// SIMATIC STEP 7 (V5.x) project ZEn01_01_STEP7__STL_1-9
// CPU: CPU314(1)
// station: _S7H_BUSSYSTEM_CT
// station: Hardware
// station: SIMATIC 300(1)
// program: S7-Program(1)

SYMBOL_TABLE
"Petrol"	DB 1	FB 1	// Data for petrol engine
"Diesel"	DB 2	FB 1	// Data for diesel engine
"S_Data"	DB 3	DB 3	// Shared data block
"Engine"	FB 1	FB 1	// Engine control
"Fan"	FC 1	FC 1	// Fan control
"Key_1"	I 0.1	BOOL	// For the AND query
"Key_2"	I 0.2	BOOL	// For the AND query
"Key_3"	I 0.3	BOOL	// For the OR query
"Key_4"	I 0.4	BOOL	// For the OR query
"Automatic_On"	I 0.5	BOOL	// For the memory function (switch on)
"Manual_On"	I 0.6	BOOL	// For the memory function (switch off)
"Switch_On_PE"	I 1.0	BOOL	// Switch on petrol engine
"Switch_Off_PE"	I 1.1	BOOL	// Switch off petrol engine
"PE_Failure"	I 1.2	BOOL	// Petrol engine failure
"Switch_On_DE"	I 1.4	BOOL	// Switch on diesel engine
"Switch_Off_DE"	I 1.5	BOOL	// Switch off diesel engine
"DE_Failure"	I 1.6	BOOL	// Diesel engine failure
"PE_Actual_Speed"	MW 2	INT	// Actual speed for petrol engine
"DE_Actual_Speed"	MW 4	INT	// Actual speed for diesel engine
"Main_Program"	OB 1	OB 1	// This block contains the user program
"Green_Light"	Q 4.0	BOOL	// Result of AND query
"Red_Light"	Q 4.1	BOOL	// Result of OR query
"Automatic_Mode"	Q 4.2	BOOL	// Retentive output
"PE_On"	Q 5.0	BOOL	// Command for switching on petrol engine
"PE_Preset_Speed_Reached"	Q 5.1	BOOL	// Display "Petrol engine preset speed reached"
"PE_Fan_On"	Q 5.2	BOOL	// Command for switching on petrol engine fan
"DE_On"	Q 5.4	BOOL	// Command for switching on diesel engine
"DE_Preset_Speed_Reached"	Q 5.5	BOOL	// Display "Diesel engine preset speed reached"
"DE_Fan_On"	Q 5.6	BOOL	// Command for switching on diesel engine fan
"PE_Follow_On"	T 1	TIMER	// Follow-on time for petrol engine fan
"DE_Follow_On"	T 2	TIMER	// Follow-on time for diesel engine fan
END_SYMBOL_TABLE

FUNCTION_BLOCK "Engine"	// FB 1
TITLE = Function Block for Controlling the Engine
//Working with STEP 7
//for the STL programming language (Statement List)
//
//Chapter 5: Creating a Program with Function Blocks and Data Blocks
//
//Description of the Function Block
//---------------------------------
//The function block contains a memory function for controlling the engine
//(a retentive output) and a comparator for monitoring 
//the speed.
//
//We want to use the same function block to control two different engines.
//We therefore want to assign all the "engine-specific" signals as block 
//parameters. The signals that are scanned are the inputs of the function 
//block ("in" declaration); the signals that are modified are the outputs 
//("out" declaration).
//
//When the function block is processed (block call) in the organization 
//block OB1, we will assign the block parameters the specific signals for 
//each engine.
//
//The operating mode (here "automatic mode") is not engine-specific; it is 
//valid for the entire control program. This signal is therefore not a 
//block parameter; it is scanned directly in the function block.
//
//Note: Only letters, numbers, and the underscore can be used for the names
//of the block parameters. In the symbol table, however, you can use all
//printable characters, including spaces and special characters.
//
AUTHOR : Siemens
FAMILY : GetStart
NAME : ENGINE
VERSION : 1.0
VAR_INPUT
  Switch_On : BOOL ;	//Switch on engine
  Switch_Off : BOOL ;	//Switch off engine
  Failure : BOOL ;	//Engine failure, causes the engine to switch off
  Actual_Speed : INT ;	//Actual engine speed
END_VAR
VAR_OUTPUT
  Engine_On : BOOL ;	//Engine is switched on
  Preset_Speed_Reached : BOOL ;	//Preset speed reached
END_VAR
VAR
  Preset_Speed : INT  := 1500;	//Requested engine speed
END_VAR
BEGIN
NETWORK
TITLE = Switching on Engine, Negating Signals
//The operations S (Set) and R (Reset) are used to switch on the engine; 
//this is the memory function.
//
//The engine is switched on when the variable #Switch_On is activated 
//(signal state "1") and the variable "Automatic_Mode" is deactivated
//(signal state "0"). The scan for signal state "0" is represented by  
//an "N" after the operation (that is, "AN").
//
//The engine is switched off again when the variable #Switch_Off is activated
//or the variable #Failure has the signal state "0". #Failure is a "zero-active"
//signal, which usually has the signal state "1" (if there is no error) and
//signal state "0" when an error occurs. Here too, we can obtain the required
//function if we scan the signal #Failure with "ON" for signal state "0". 
//
//Note: "Block-specific" variables are represented with a hash symbol before
//the name (#name) and are only valid within the block. Shared variables
//appear in quotation marks ("name") and are valid in the entire program.
      A     #Switch_On;
      AN    "Automatic_Mode";
      S     #Engine_On;
      O     #Switch_Off;
      ON    #Failure;
      R     #Engine_On;
NETWORK
TITLE = Monitoring the Speed
//A comparator monitors the engine speed. It checks whether the actual speed
//is greater than or equal to the preset speed. If this is the case, the 
//comparator sets the variable #Preset_Speed_Reached.
//
//The variables to be compared are loaded into the internal registers using
//the load instruction "L". Then, the instruction ">=I" compares the contents
//of the internal registers (here, for greater than or equal to with number
//format INTEGER) and supplies a binary comparison result. This is assigned 
//to the variable #Preset_Speed_Reached.
//
//The actual engine speed is a block input parameter ("in" declaration), 
//because it is engine-specific. The preset speed is also engine-specific, 
//but because it is a fixed value, it can be stored as static data in the engine  
//data ("stat" declaration). This is known as a "static local variable."
      L     #Actual_Speed;
      L     #Preset_Speed;
      >=I;
      =     #Preset_Speed_Reached;
END_FUNCTION_BLOCK

FUNCTION "Fan" : VOID	// FC 1
TITLE = Function for Controlling the Fan
//Working with STEP 7
//for the STL programming language (Statement List)
//
//Chapter 8: Programming a Function 
//
//Description of the Function
//---------------------------
//You can program a function (FC) when the algorithm (the control function)
//does not have to store any of its own data. In contrast to a function 
//block (FB), a function has no instance data block.
//
//The example shows a simple function: a fan starts when the engine is 
//switched on. When the engine is switched off again, the fan continues to 
//run for another 4 seconds and then stops.
//
AUTHOR : Siemens
FAMILY : GetStart
NAME : FAN
VERSION : 1.0
VAR_INPUT
  Engine_On : BOOL ;	//Signal for switching on the engine
  Timer_Function : TIMER ;	//Timer function used for the switch-off delay
END_VAR
VAR_OUTPUT
  Fan_On : BOOL ;	//Signal for switching on the fan
END_VAR
BEGIN
NETWORK
TITLE = Controlling the fan
//The variable #Timer_Function is started with the input parameter #Engine_On. 
//via the instruction SF (start time as switch-off delay). This variable 
//#Timer_Function with the data type TIMER stands for a timer function which,
//is assigned a timer address (for example, T1) later on when it is called in 
//OB1. You must select a different timer address for each engine fan pair every 
//time you call the timer function.
//
//A constant switch-off delay of 4 seconds is loaded before starting the timer. 
//function. You can also assign the time delay as an input parameter with the 
//data type S5TIME so that a different follow-on time can be configured for the 
//fan in each engine. 
      A     #Engine_On;
      L     S5T#4S;
      SF    #Timer_Function;
      A     #Timer_Function;
      =     #Fan_On;
END_FUNCTION

DATA_BLOCK "Petrol"	// DB 1
AUTHOR : Siemens
FAMILY : GetStart
NAME : Petrol
VERSION : 1.0
"Engine"
BEGIN
END_DATA_BLOCK

DATA_BLOCK "Diesel"	// DB 2
AUTHOR : Siemens
FAMILY : GetStart
NAME : Diesel
VERSION : 1.0
"Engine"
BEGIN
END_DATA_BLOCK

DATA_BLOCK "S_Data"	// DB 3
AUTHOR : Siemens
FAMILY : GetStart
NAME : S_Data
VERSION : 1.0
  STRUCT
   PE_Actual_Speed : INT ;	//Actual speed for petrol engine
   DE_Actual_Speed : INT ;	//Actual speed for petrol engine
   Preset_Speed_Reached : BOOL ;	//Both engines have reached the preset speed
  END_STRUCT ;	
BEGIN
END_DATA_BLOCK

ORGANIZATION_BLOCK "Main_Program"	// OB 1
TITLE = Cyclically Processed Main Program
//Working with STEP 7
//for the STL programming language (Statement List)
//
//Chapter 4: Creating a Program in OB1 (Networks 1 to 3)
//Chapter 5: Creating a Program with Function Blocks and Data Blocks (Networks 4 
//and 5)
//Chapter 8: Programming a Function (Networks 6 and 7)
//
AUTHOR : Siemens
FAMILY : GetStart
NAME : Cycle
VERSION : 1.0
VAR_TEMP
  OB1_EV_CLASS : BYTE ;	//Bits 0 to 3 = 1 (incoming event), bits 4 to 7 = 1 (event class 1)
  OB1_SCAN_1 : BYTE ;	//1 (cold restart scan 1 of OB1), 3 (Scan 2-n of OB1)
  OB1_PRIORITY : BYTE ;	//1 (priority of 1 is lowest)
  OB1_OB_NUMBR : BYTE ;	//1 (organization block 1, OB1)
  OB1_RESERVED_1 : BYTE ;	//Reserved for system
  OB1_RESERVED_2 : BYTE ;	//Reserved for system
  OB1_PREV_CYCLE : INT ;	//Cycle time of previous OB1 scan (milliseconds)
  OB1_MIN_CYCLE : INT ;	//Minimum cycle time of OB1 (milliseconds)
  OB1_MAX_CYCLE : INT ;	//Maximum cycle time of OB1 (milliseconds)
  OB1_DATE_TIME : DATE_AND_TIME ;	//Date and time OB1 started
END_VAR
BEGIN
NETWORK
TITLE = AND Scan
//When both "Key 1" (I 0.1) and "Key 2" (I 0.2) are activated 
//(that is, they have the signal state "1" = 24 V), the "Green Light" (Q 4.0) 
//is activated.
//
//Both inputs must be activated in order for the lamp to switch on.
      A     "Key_1";
      A     "Key_2";
      =     "Green_Light";
NETWORK
TITLE = OR Scan
//When either "Key 3" (I 0.3) or "Key 4" (I 0.4) is activated
//(that is, one has the signal state "1" = 24 V), the "Red Light" (Q 4.1)
//is activated.
//
//Only one of the inputs needs to be activated in order for the lamp to switch 
//on.
      O     "Key_3";
      O     "Key_4";
      =     "Red_Light";
NETWORK
TITLE = Retentive Activating and Deactivating
//When "Automatic On" (I 0.5) is activated, "Automatic_Mode" (Q 4.2) is also 
//activated using the operation S and remains active even if "Automatic On" 
//(I 0.5) is deactivated again.
//
//When "Manual On" (I 0.6) is activated, "Automatic Mode" (Q 4.2) is deactivated 
//again using the operation R and remains deactivated even if "Manual On" (I 0.6) 
//is deactivated again.
//
//The signal state is stored with the operations S (Set) and R (Reset). 
//If you activate both inputs simultaneously, first the set function and then
//the reset function is processed. Due to the programming sequence the reset 
//function "wins" in the end: "Automatic On" (Q 4.2) is or remains deactivated. 
//In this case, we say "Resetting has first priority".
      A     "Automatic_On";
      S     "Automatic_Mode";
      A     "Manual_On";
      R     "Automatic_Mode";
NETWORK
TITLE = Switching on the Petrol Engine
//Call for the function block FB1 ("Engine") with the data for a 
//petrol engine (data block "Petrol" DB1).
      CALL  "Engine" , "Petrol" (
           Switch_On                := "Switch_On_PE",
           Switch_Off               := "Switch_Off_PE",
           Failure                  := "PE_Failure",
           Actual_Speed             := "PE_Actual_Speed",
           Engine_On                := "PE_On",
           Preset_Speed_Reached     := "PE_Preset_Speed_Reached");
NETWORK
TITLE = Switching on the Diesel Engine
//Call for the function block FB1 ("Engine") with the data for a
//diesel engine (data block "Diesel" DB2).
      CALL  "Engine" , "Diesel" (
           Switch_On                := "Switch_On_DE",
           Switch_Off               := "Switch_Off_DE",
           Failure                  := "DE_Failure",
           Actual_Speed             := "DE_Actual_Speed",
           Engine_On                := "DE_On",
           Preset_Speed_Reached     := "DE_Preset_Speed_Reached");
NETWORK
TITLE = Controlling the Fan for the Petrol Engine
//Call for the function FC1 for the petrol engine.
      CALL  "Fan" (
           Engine_On                := "PE_On",
           Timer_Function           := "PE_Follow_On",
           Fan_On                   := "PE_Fan_On");
NETWORK
TITLE = Controlling the Fan for the Diesel Engine
//Call for the function FC1 for the diesel engine.
      CALL  "Fan" (
           Engine_On                := "DE_On",
           Timer_Function           := "DE_Follow_On",
           Fan_On                   := "DE_Fan_On");
END_ORGANIZATION_BLOCK
